FUNCTION F_ConfigDataTypeSize : UDINT
VAR_INPUT
	DataType : E_ConfigDataType;
END_VAR

CASE DataType OF
	E_ConfigDataType.Boolean:
		F_ConfigDataTypeSize := SIZEOF(BOOL);
	E_ConfigDataType.Integer32:
		F_ConfigDataTypeSize := SIZEOF(DINT);
	E_ConfigDataType.UnsignedInteger32:
		F_ConfigDataTypeSize := SIZEOF(UDINT);
	E_ConfigDataType.Float32:
		F_ConfigDataTypeSize := SIZEOF(REAL);
	E_ConfigDataType.Float64:
		F_ConfigDataTypeSize := SIZEOF(LREAL);
	E_ConfigDataType.String80:
		F_ConfigDataTypeSize := 81;
ELSE
	F_ConfigDataTypeSize := 0;
END_CASE

END_FUNCTION

(* stored: Version 1.1.0.1, ProductVersion 3.1.4026.18
   POU F_ConfigDataTypeSize: Id {77fcb289-6570-44ba-9a67-58620a6f624d}, SpecialFunc None *)
